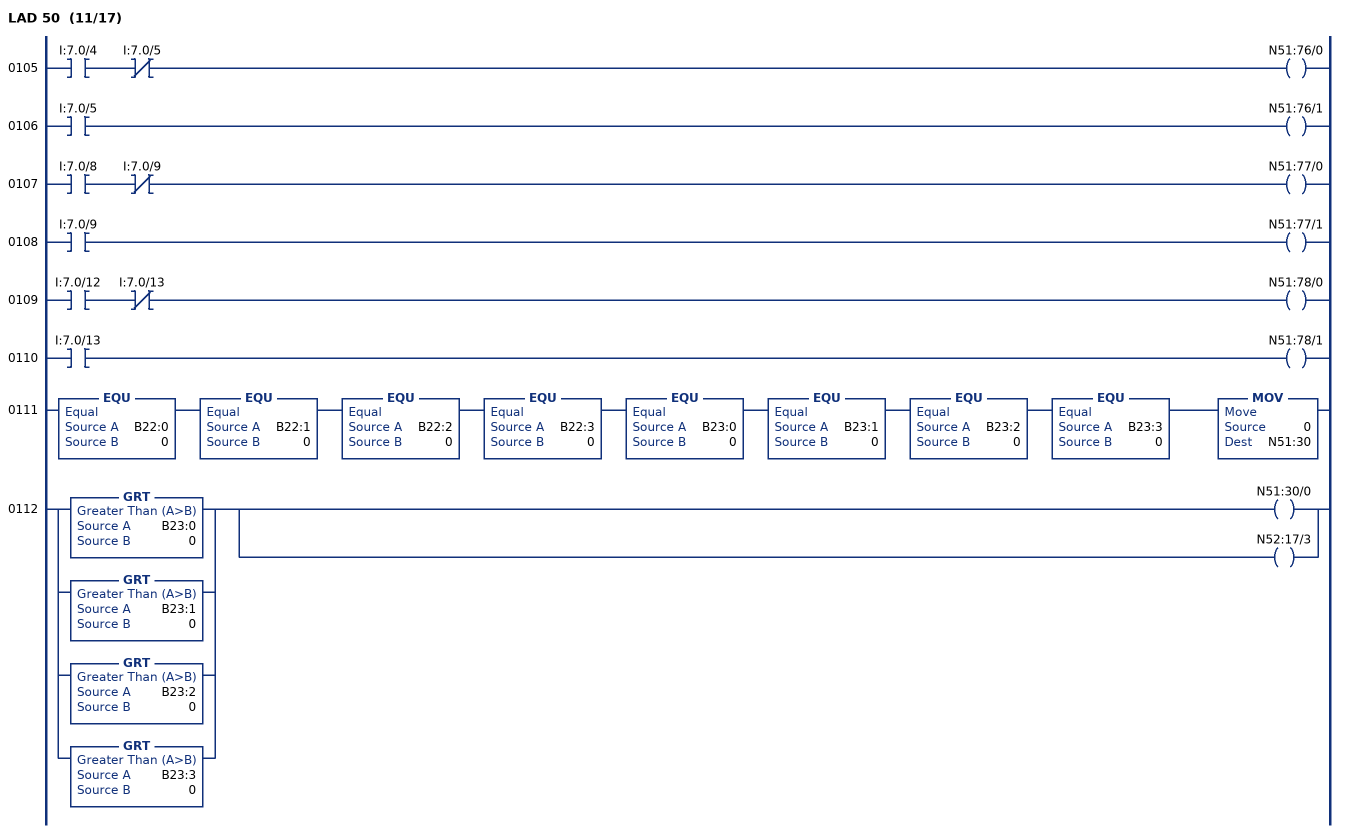
% Rung: 105 %
SOR XIC I:7.0/4 XIO I:7.0/5 OTE N51:76/0 EOR
% Rung: 106 %
SOR XIC I:7.0/5 OTE N51:76/1 EOR
% Rung: 107 %
SOR XIC I:7.0/8 XIO I:7.0/9 OTE N51:77/0 EOR
% Rung: 108 %
SOR XIC I:7.0/9 OTE N51:77/1 EOR
% Rung: 109 %
SOR XIC I:7.0/12 XIO I:7.0/13 OTE N51:78/0 EOR
% Rung: 110 %
SOR XIC I:7.0/13 OTE N51:78/1 EOR
% Rung: 111 %
SOR EQU B22:0 0 EQU B22:1 0 EQU B22:2 0 EQU B22:3 0 EQU B23:0 0 EQU B23:1 0 EQU B23:2 0 EQU B23:3 0 MOV 0 N51:30 EOR
% Rung: 112 %
SOR BST GRT B23:0 0 NXB GRT B23:1 0 NXB GRT B23:2 0 NXB GRT B23:3 0 BND BST OTE N51:30/0 NXB OTE N52:17/3 BND EOR

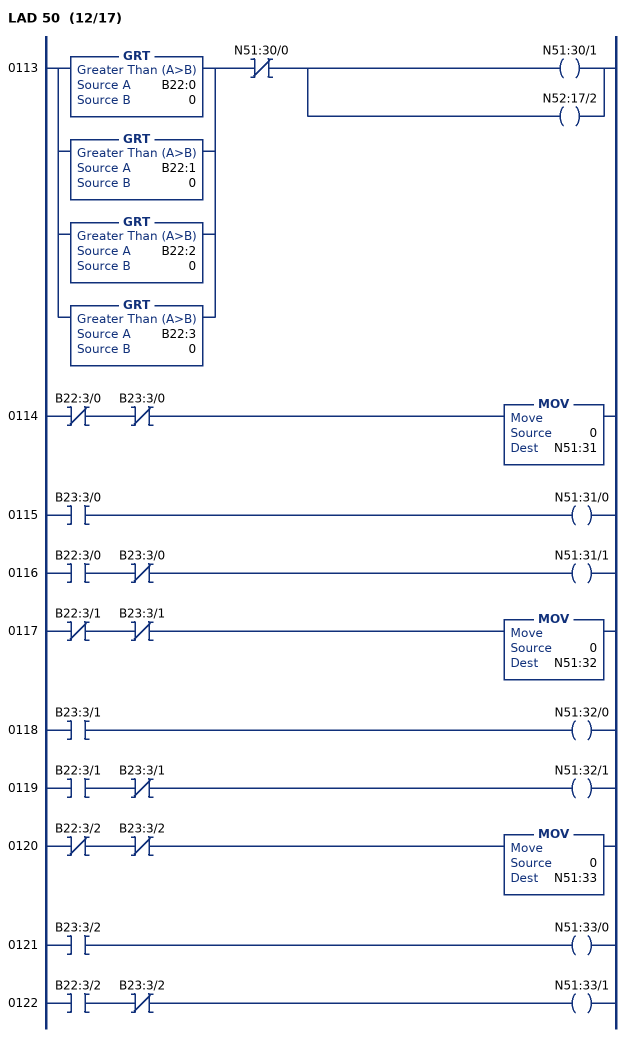
% Rung: 113 %
SOR BST GRT B22:0 0 NXB GRT B22:1 0 NXB GRT B22:2 0 NXB GRT B22:3 0 BND XIO N51:30/0 BST OTE N51:30/1 NXB OTE N52:17/2 BND EOR
% Rung: 114 %
SOR XIO B22:3/0 XIO B23:3/0 MOV 0 N51:31 EOR
% Rung: 115 %
SOR XIC B23:3/0 OTE N51:31/0 EOR
% Rung: 116 %
SOR XIC B22:3/0 XIO B23:3/0 OTE N51:31/1 EOR
% Rung: 117 %
SOR XIO B22:3/1 XIO B23:3/1 MOV 0 N51:32 EOR
% Rung: 118 %
SOR XIC B23:3/1 OTE N51:32/0 EOR
% Rung: 119 %
SOR XIC B22:3/1 XIO B23:3/1 OTE N51:32/1 EOR
% Rung: 120 %
SOR XIO B22:3/2 XIO B23:3/2 MOV 0 N51:33 EOR
% Rung: 121 %
SOR XIC B23:3/2 OTE N51:33/0 EOR
% Rung: 122 %
SOR XIC B22:3/2 XIO B23:3/2 OTE N51:33/1 EOR

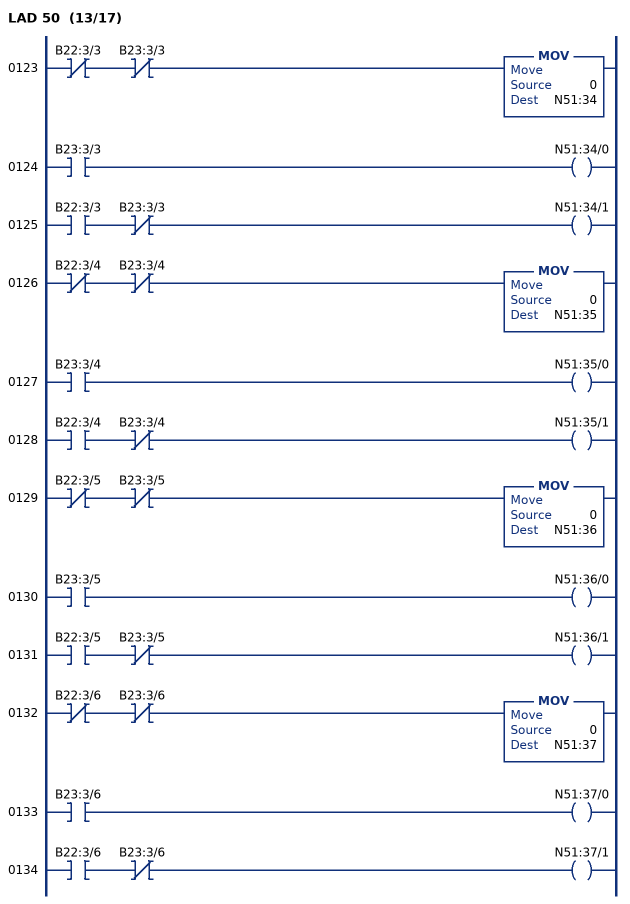
% Rung: 123 %
SOR XIO B22:3/3 XIO B23:3/3 MOV 0 N51:34 EOR
% Rung: 124 %
SOR XIC B23:3/3 OTE N51:34/0 EOR
% Rung: 125 %
SOR XIC B22:3/3 XIO B23:3/3 OTE N51:34/1 EOR
% Rung: 126 %
SOR XIO B22:3/4 XIO B23:3/4 MOV 0 N51:35 EOR
% Rung: 127 %
SOR XIC B23:3/4 OTE N51:35/0 EOR
% Rung: 128 %
SOR XIC B22:3/4 XIO B23:3/4 OTE N51:35/1 EOR
% Rung: 129 %
SOR XIO B22:3/5 XIO B23:3/5 MOV 0 N51:36 EOR
% Rung: 130 %
SOR XIC B23:3/5 OTE N51:36/0 EOR
% Rung: 131 %
SOR XIC B22:3/5 XIO B23:3/5 OTE N51:36/1 EOR
% Rung: 132 %
SOR XIO B22:3/6 XIO B23:3/6 MOV 0 N51:37 EOR
% Rung: 133 %
SOR XIC B23:3/6 OTE N51:37/0 EOR
% Rung: 134 %
SOR XIC B22:3/6 XIO B23:3/6 OTE N51:37/1 EOR

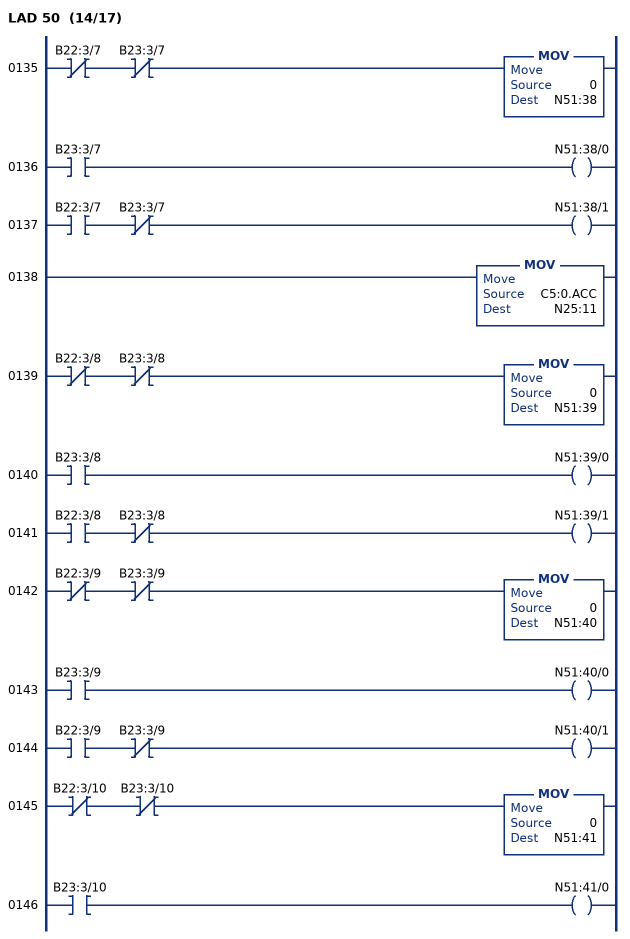
% Rung: 135 %
SOR XIO B22:3/7 XIO B23:3/7 MOV 0 N51:38 EOR
% Rung: 136 %
SOR XIC B23:3/7 OTE N51:38/0 EOR
% Rung: 137 %
SOR XIC B22:3/7 XIO B23:3/7 OTE N51:38/1 EOR
% Rung: 138 %
SOR MOV C5:0.ACC N25:11 EOR
% Rung: 139 %
SOR XIO B22:3/8 XIO B23:3/8 MOV 0 N51:39 EOR
% Rung: 140 %
SOR XIC B23:3/8 OTE N51:39/0 EOR
% Rung: 141 %
SOR XIC B22:3/8 XIO B23:3/8 OTE N51:39/1 EOR
% Rung: 142 %
SOR XIO B22:3/9 XIO B23:3/9 MOV 0 N51:40 EOR
% Rung: 143 %
SOR XIC B23:3/9 OTE N51:40/0 EOR
% Rung: 144 %
SOR XIC B22:3/9 XIO B23:3/9 OTE N51:40/1 EOR
% Rung: 145 %
SOR XIO B22:3/10 XIO B23:3/10 MOV 0 N51:41 EOR
% Rung: 146 %
SOR XIC B23:3/10 OTE N51:41/0 EOR

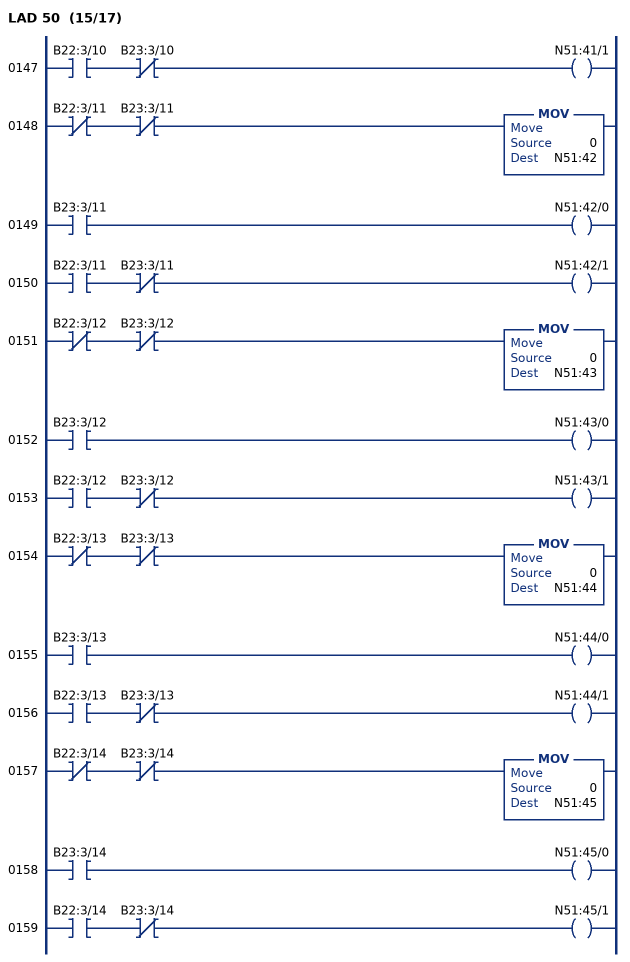
% Rung: 147 %
SOR XIC B22:3/10 XIO B23:3/10 OTE N51:41/1 EOR
% Rung: 148 %
SOR XIO B22:3/11 XIO B23:3/11 MOV 0 N51:42 EOR
% Rung: 149 %
SOR XIC B23:3/11 OTE N51:42/0 EOR
% Rung: 150 %
SOR XIC B22:3/11 XIO B23:3/11 OTE N51:42/1 EOR
% Rung: 151 %
SOR XIO B22:3/12 XIO B23:3/12 MOV 0 N51:43 EOR
% Rung: 152 %
SOR XIC B23:3/12 OTE N51:43/0 EOR
% Rung: 153 %
SOR XIC B22:3/12 XIO B23:3/12 OTE N51:43/1 EOR
% Rung: 154 %
SOR XIO B22:3/13 XIO B23:3/13 MOV 0 N51:44 EOR
% Rung: 155 %
SOR XIC B23:3/13 OTE N51:44/0 EOR
% Rung: 156 %
SOR XIC B22:3/13 XIO B23:3/13 OTE N51:44/1 EOR
% Rung: 157 %
SOR XIO B22:3/14 XIO B23:3/14 MOV 0 N51:45 EOR
% Rung: 158 %
SOR XIC B23:3/14 OTE N51:45/0 EOR
% Rung: 159 %
SOR XIC B22:3/14 XIO B23:3/14 OTE N51:45/1 EOR

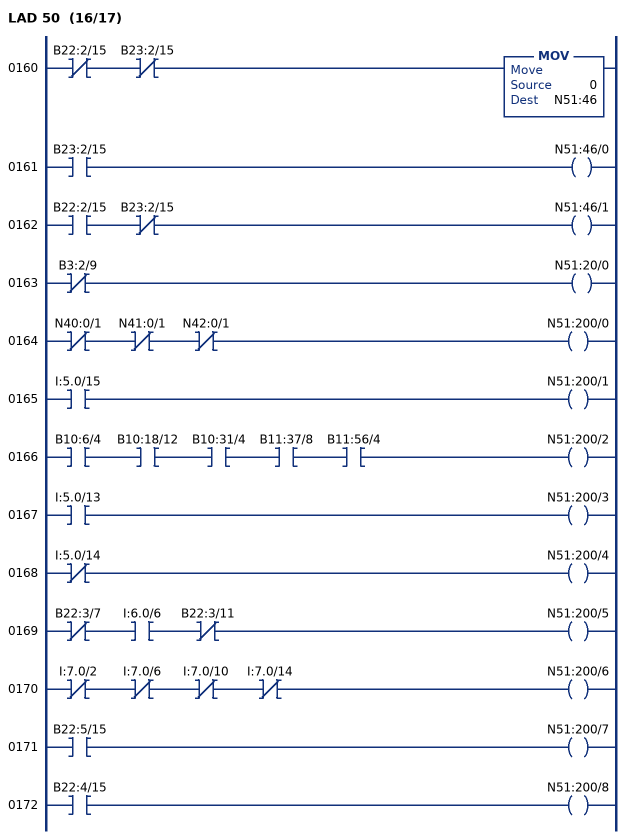
% Rung: 160 %
SOR XIO B22:2/15 XIO B23:2/15 MOV 0 N51:46 EOR
% Rung: 161 %
SOR XIC B23:2/15 OTE N51:46/0 EOR
% Rung: 162 %
SOR XIC B22:2/15 XIO B23:2/15 OTE N51:46/1 EOR
% Rung: 163 %
SOR XIO B3:2/9 OTE N51:20/0 EOR
% Rung: 164 %
SOR XIO N40:0/1 XIO N41:0/1 XIO N42:0/1 OTE N51:200/0 EOR
% Rung: 165 %
SOR XIC I:5.0/15 OTE N51:200/1 EOR
% Rung: 166 %
SOR XIC B10:6/4 XIC B10:18/12 XIC B10:31/4 XIC B11:37/8 XIC B11:56/4 OTE N51:200/2 EOR
% Rung: 167 %
SOR XIC I:5.0/13 OTE N51:200/3 EOR
% Rung: 168 %
SOR XIO I:5.0/14 OTE N51:200/4 EOR
% Rung: 169 %
SOR XIO B22:3/7 XIC I:6.0/6 XIO B22:3/11 OTE N51:200/5 EOR
% Rung: 170 %
SOR XIO I:7.0/2 XIO I:7.0/6 XIO I:7.0/10 XIO I:7.0/14 OTE N51:200/6 EOR
% Rung: 171 %
SOR XIC B22:5/15 OTE N51:200/7 EOR
% Rung: 172 %
SOR XIC B22:4/15 OTE N51:200/8 EOR

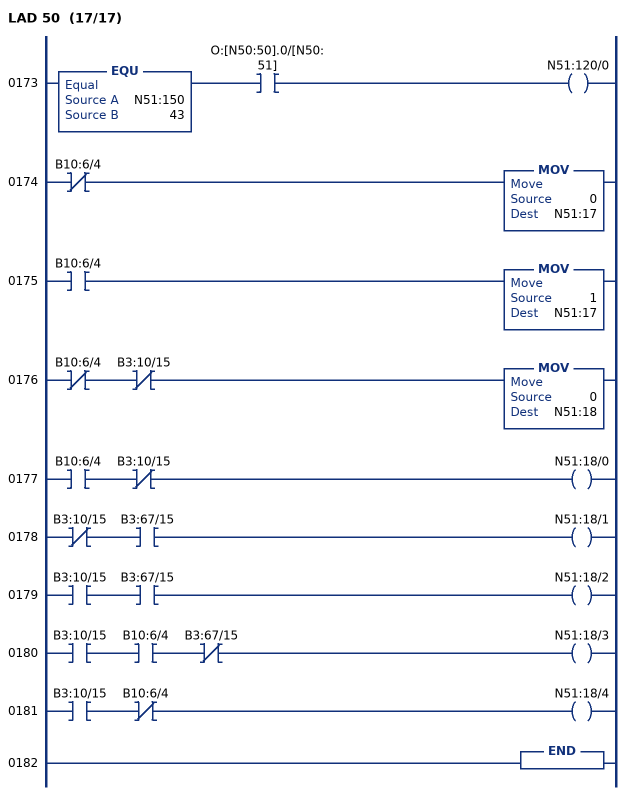
% Rung: 173 %
SOR EQU N51:150 43 XIC O:[N50:50].0/[N50:51] OTE N51:120/0 EOR
% Rung: 174 %
SOR XIO B10:6/4 MOV 0 N51:17 EOR
% Rung: 175 %
SOR XIC B10:6/4 MOV 1 N51:17 EOR
% Rung: 176 %
SOR XIO B10:6/4 XIO B3:10/15 MOV 0 N51:18 EOR
% Rung: 177 %
SOR XIC B10:6/4 XIO B3:10/15 OTE N51:18/0 EOR
% Rung: 178 %
SOR XIO B3:10/15 XIC B3:67/15 OTE N51:18/1 EOR
% Rung: 179 %
SOR XIC B3:10/15 XIC B3:67/15 OTE N51:18/2 EOR
% Rung: 180 %
SOR XIC B3:10/15 XIC B10:6/4 XIO B3:67/15 OTE N51:18/3 EOR
% Rung: 181 %
SOR XIC B3:10/15 XIO B10:6/4 OTE N51:18/4 EOR
% Rung: 182 %
SOR END EOR

LADDER 51
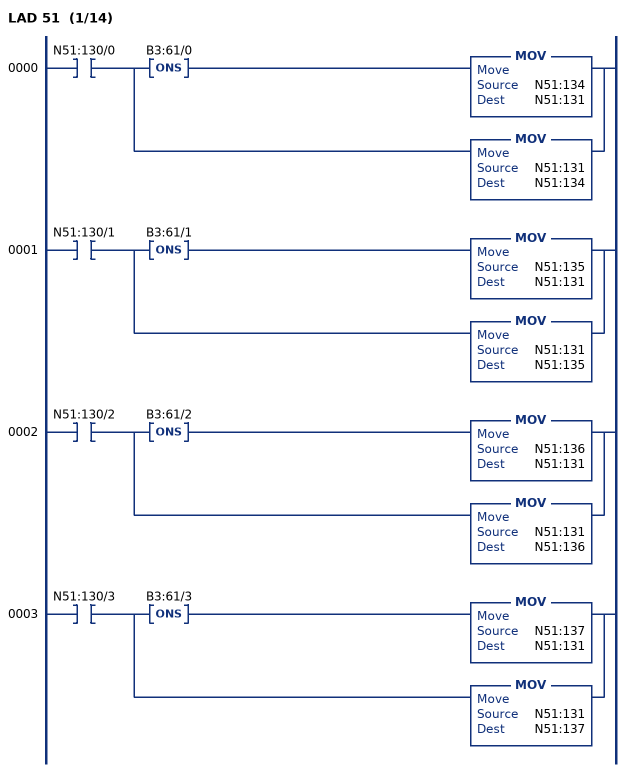
% Rung: 0 %
SOR XIC N51:130/0 BST OSR B3:61/0 MOV N51:134 N51:131 NXB MOV N51:131 N51:134 BND EOR
% Rung: 1 %
SOR XIC N51:130/1 BST OSR B3:61/1 MOV N51:135 N51:131 NXB MOV N51:131 N51:135 BND EOR
% Rung: 2 %
SOR XIC N51:130/2 BST OSR B3:61/2 MOV N51:136 N51:131 NXB MOV N51:131 N51:136 BND EOR
% Rung: 3 %
SOR XIC N51:130/3 BST OSR B3:61/3 MOV N51:137 N51:131 NXB MOV N51:131 N51:137 BND EOR

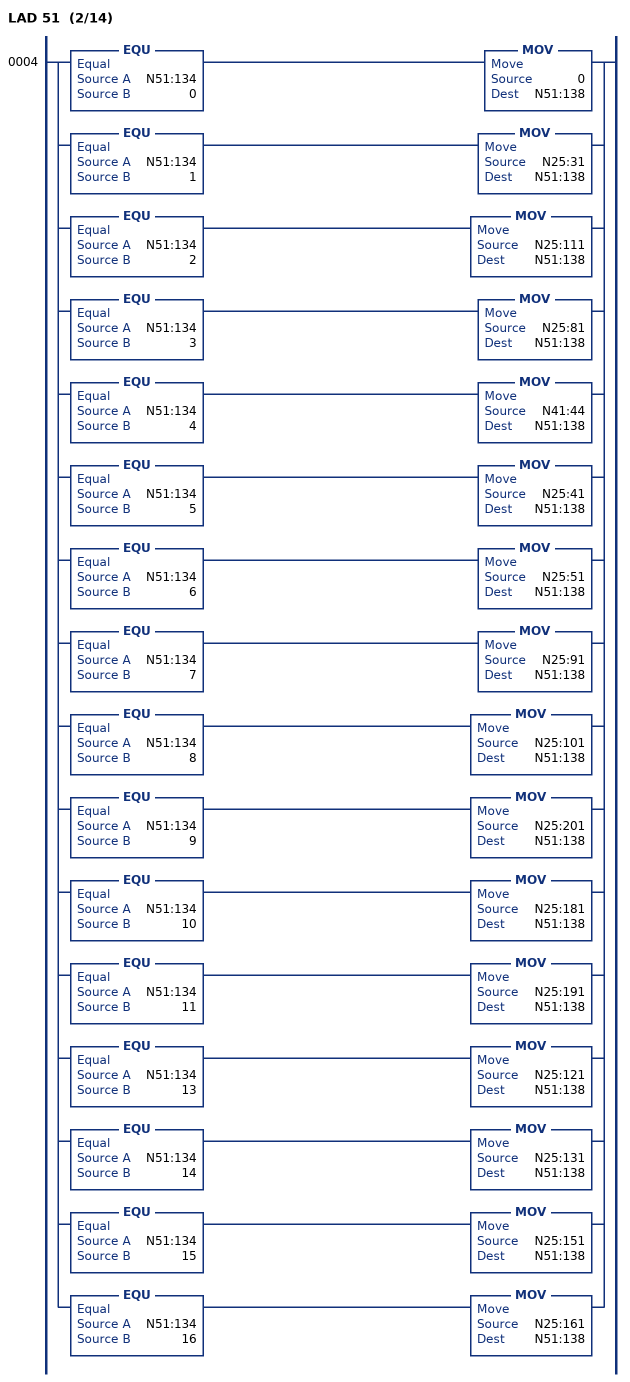
% Rung: 4 %
SOR BST EQU N51:134 0 MOV 0 N51:138 NXB EQU N51:134 1 MOV N25:31 N51:138 NXB EQU N51:134 2 MOV N25:111 N51:138 NXB EQU N51:134 3 MOV N25:81 N51:138 NXB EQU N51:134 4 MOV N41:44 N51:138 NXB EQU N51:134 5 MOV N25:41 N51:138 NXB EQU N51:134 6 MOV N25:51 N51:138 NXB EQU N51:134 7 MOV N25:91 N51:138 NXB EQU N51:134 8 MOV N25:101 N51:138 NXB EQU N51:134 9 MOV N25:201 N51:138 NXB EQU N51:134 10 MOV N25:181 N51:138 NXB EQU N51:134 11 MOV N25:191 N51:138 NXB EQU N51:134 13 MOV N25:121 N51:138 NXB EQU N51:134 14 MOV N25:131 N51:138 NXB EQU N51:134 15 MOV N25:151 N51:138 NXB EQU N51:134 16 MOV N25:161 N51:138 BND EOR

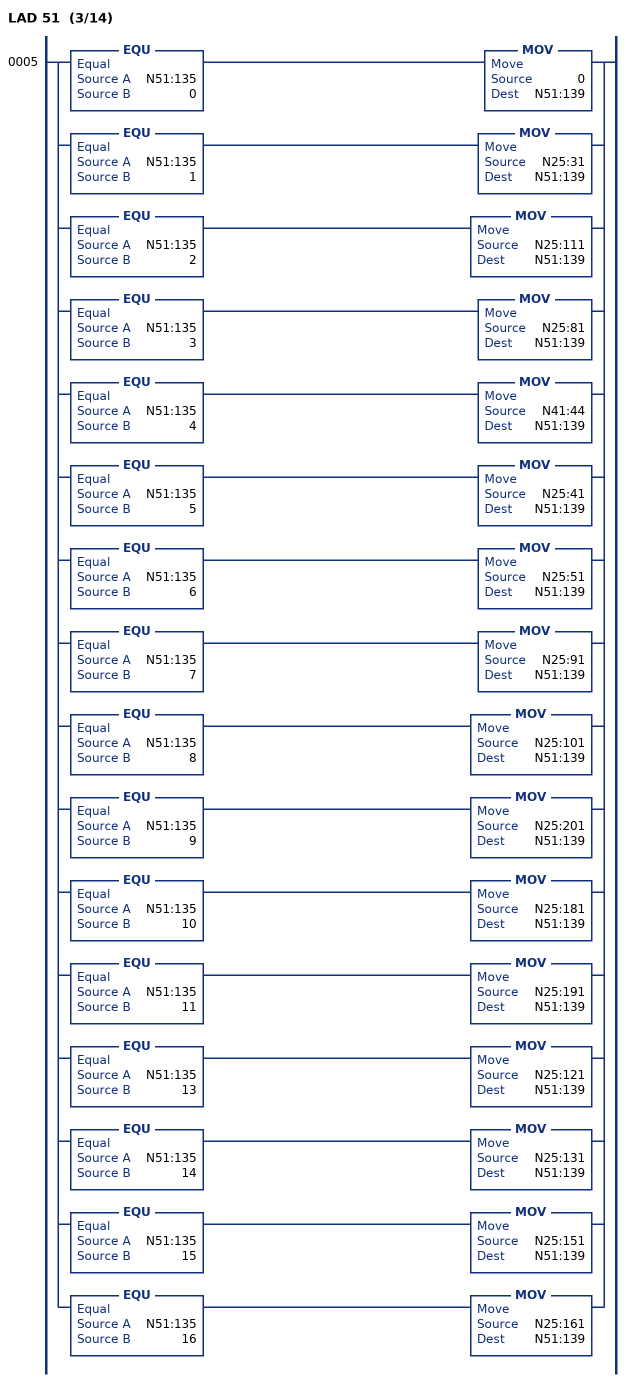
% Rung: 5 %
SOR BST EQU N51:135 0 MOV 0 N51:139 NXB EQU N51:135 1 MOV N25:31 N51:139 NXB EQU N51:135 2 MOV N25:111 N51:139 NXB EQU N51:135 3 MOV N25:81 N51:139 NXB EQU N51:135 4 MOV N41:44 N51:139 NXB EQU N51:135 5 MOV N25:41 N51:139 NXB EQU N51:135 6 MOV N25:51 N51:139 NXB EQU N51:135 7 MOV N25:91 N51:139 NXB EQU N51:135 8 MOV N25:101 N51:139 NXB EQU N51:135 9 MOV N25:201 N51:139 NXB EQU N51:135 10 MOV N25:181 N51:139 NXB EQU N51:135 11 MOV N25:191 N51:139 NXB EQU N51:135 13 MOV N25:121 N51:139 NXB EQU N51:135 14 MOV N25:131 N51:139 NXB EQU N51:135 15 MOV N25:151 N51:139 NXB EQU N51:135 16 MOV N25:161 N51:139 BND EOR

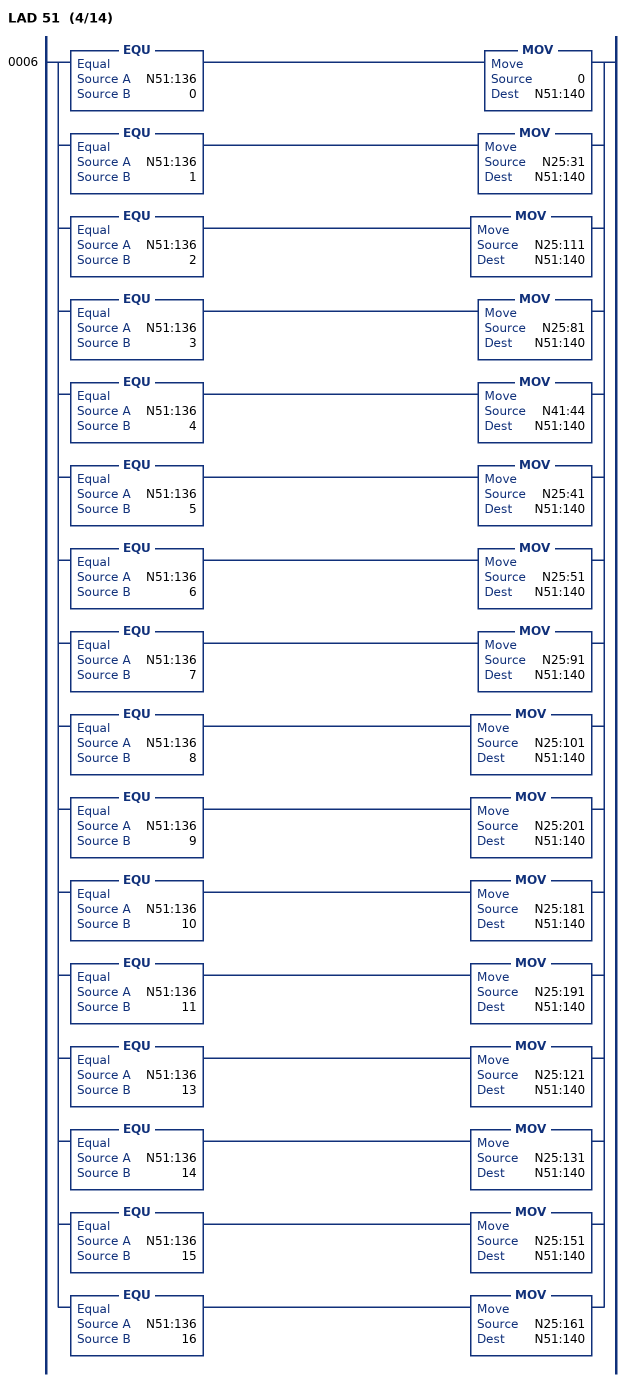
% Rung: 6 %
SOR BST EQU N51:136 0 MOV 0 N51:140 NXB EQU N51:136 1 MOV N25:31 N51:140 NXB EQU N51:136 2 MOV N25:111 N51:140 NXB EQU N51:136 3 MOV N25:81 N51:140 NXB EQU N51:136 4 MOV N41:44 N51:140 NXB EQU N51:136 5 MOV N25:41 N51:140 NXB EQU N51:136 6 MOV N25:51 N51:140 NXB EQU N51:136 7 MOV N25:91 N51:140 NXB EQU N51:136 8 MOV N25:101 N51:140 NXB EQU N51:136 9 MOV N25:201 N51:140 NXB EQU N51:136 10 MOV N25:181 N51:140 NXB EQU N51:136 11 MOV N25:191 N51:140 NXB EQU N51:136 13 MOV N25:121 N51:140 NXB EQU N51:136 14 MOV N25:131 N51:140 NXB EQU N51:136 15 MOV N25:151 N51:140 NXB EQU N51:136 16 MOV N25:161 N51:140 BND EOR

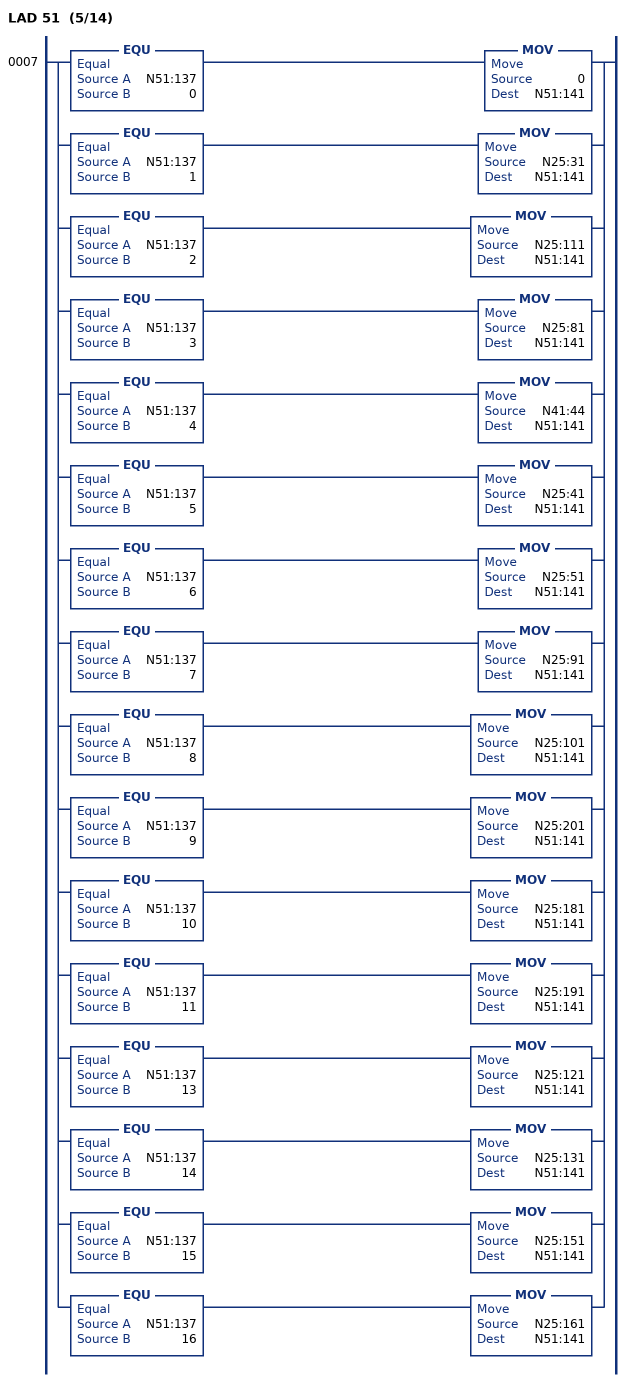
% Rung: 7 %
SOR BST EQU N51:137 0 MOV 0 N51:141 NXB EQU N51:137 1 MOV N25:31 N51:141 NXB EQU N51:137 2 MOV N25:111 N51:141 NXB EQU N51:137 3 MOV N25:81 N51:141 NXB EQU N51:137 4 MOV N41:44 N51:141 NXB EQU N51:137 5 MOV N25:41 N51:141 NXB EQU N51:137 6 MOV N25:51 N51:141 NXB EQU N51:137 7 MOV N25:91 N51:141 NXB EQU N51:137 8 MOV N25:101 N51:141 NXB EQU N51:137 9 MOV N25:201 N51:141 NXB EQU N51:137 10 MOV N25:181 N51:141 NXB EQU N51:137 11 MOV N25:191 N51:141 NXB EQU N51:137 13 MOV N25:121 N51:141 NXB EQU N51:137 14 MOV N25:131 N51:141 NXB EQU N51:137 15 MOV N25:151 N51:141 NXB EQU N51:137 16 MOV N25:161 N51:141 BND EOR

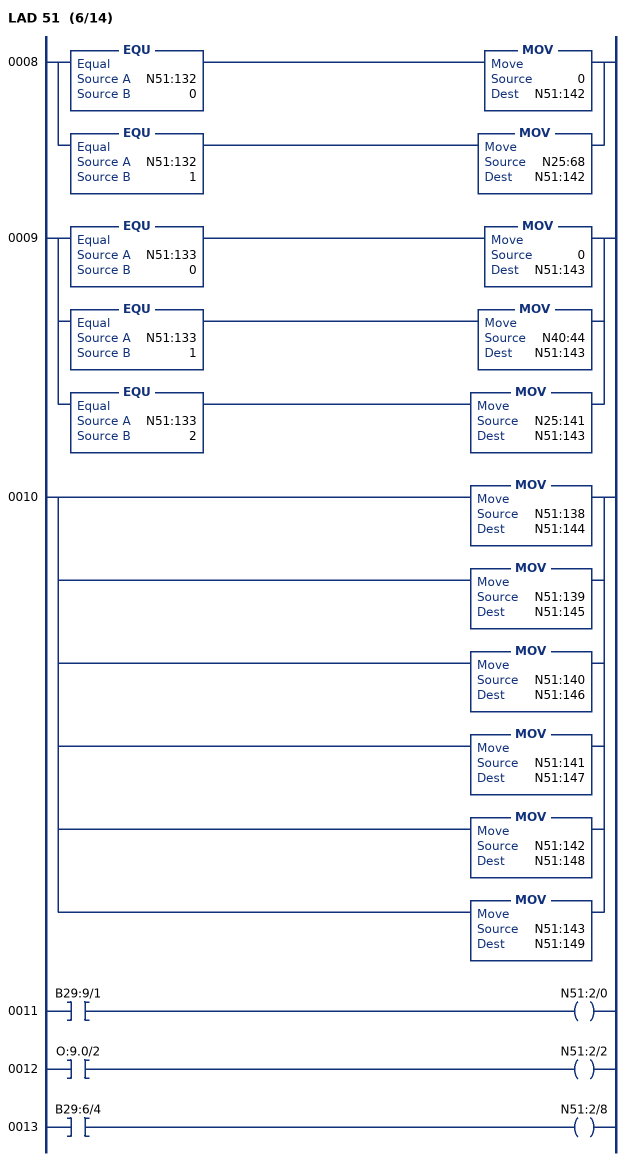
% Rung: 8 %
SOR BST EQU N51:132 0 MOV 0 N51:142 NXB EQU N51:132 1 MOV N25:68 N51:142 BND EOR
% Rung: 9 %
SOR BST EQU N51:133 0 MOV 0 N51:143 NXB EQU N51:133 1 MOV N40:44 N51:143 NXB EQU N51:133 2 MOV N25:141 N51:143 BND EOR
% Rung: 10 %
SOR BST MOV N51:138 N51:144 NXB MOV N51:139 N51:145 NXB MOV N51:140 N51:146 NXB MOV N51:141 N51:147 NXB MOV N51:142 N51:148 NXB MOV N51:143 N51:149 BND EOR
% Rung: 11 %
SOR XIC B29:9/1 OTE N51:2/0 EOR
% Rung: 12 %
SOR XIC O:9.0/2 OTE N51:2/2 EOR
% Rung: 13 %
SOR XIC B29:6/4 OTE N51:2/8 EOR

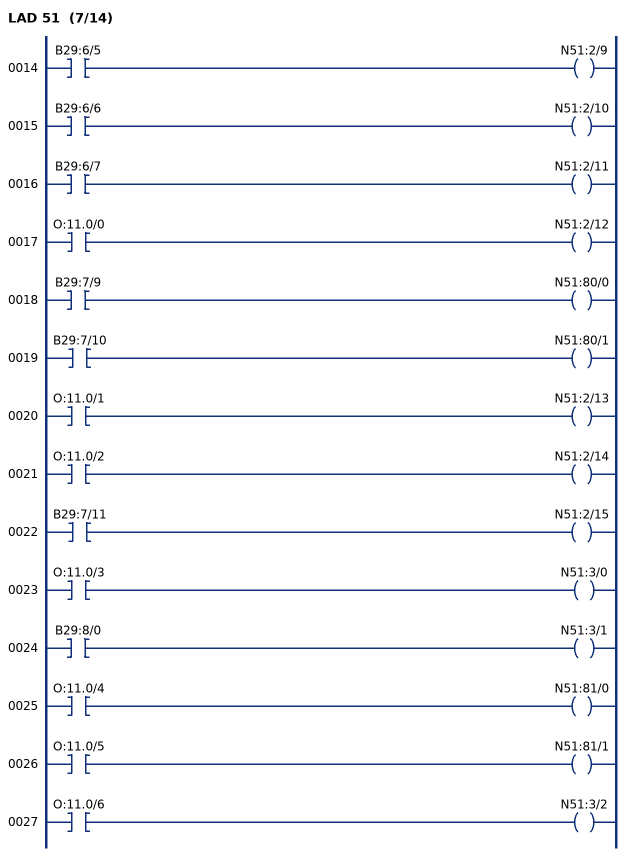
% Rung: 14 %
SOR XIC B29:6/5 OTE N51:2/9 EOR
% Rung: 15 %
SOR XIC B29:6/6 OTE N51:2/10 EOR
% Rung: 16 %
SOR XIC B29:6/7 OTE N51:2/11 EOR
% Rung: 17 %
SOR XIC O:11.0/0 OTE N51:2/12 EOR
% Rung: 18 %
SOR XIC B29:7/9 OTE N51:80/0 EOR
% Rung: 19 %
SOR XIC B29:7/10 OTE N51:80/1 EOR
% Rung: 20 %
SOR XIC O:11.0/1 OTE N51:2/13 EOR
% Rung: 21 %
SOR XIC O:11.0/2 OTE N51:2/14 EOR
% Rung: 22 %
SOR XIC B29:7/11 OTE N51:2/15 EOR
% Rung: 23 %
SOR XIC O:11.0/3 OTE N51:3/0 EOR
% Rung: 24 %
SOR XIC B29:8/0 OTE N51:3/1 EOR
% Rung: 25 %
SOR XIC O:11.0/4 OTE N51:81/0 EOR
% Rung: 26 %
SOR XIC O:11.0/5 OTE N51:81/1 EOR
% Rung: 27 %
SOR XIC O:11.0/6 OTE N51:3/2 EOR

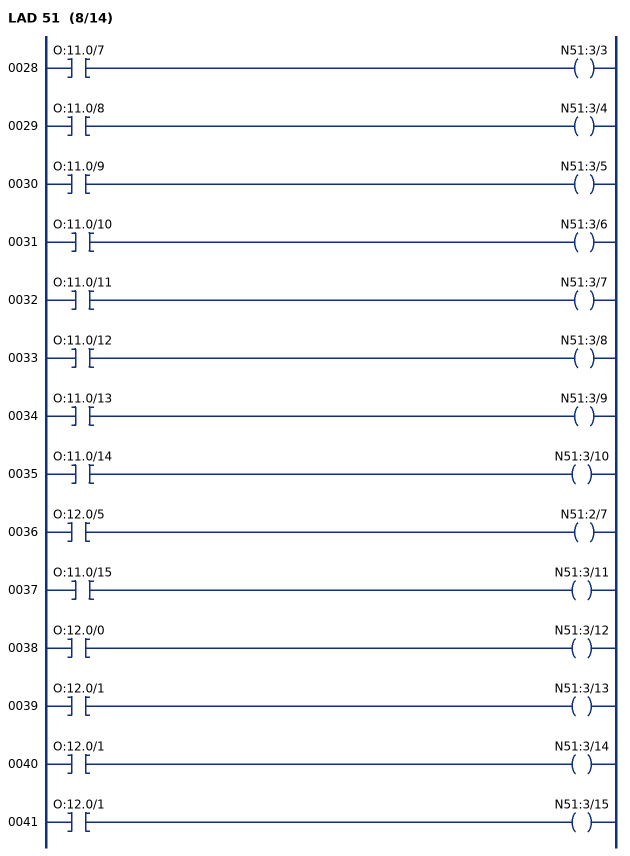
% Rung: 28 %
SOR XIC O:11.0/7 OTE N51:3/3 EOR
% Rung: 29 %
SOR XIC O:11.0/8 OTE N51:3/4 EOR
% Rung: 30 %
SOR XIC O:11.0/9 OTE N51:3/5 EOR
% Rung: 31 %
SOR XIC O:11.0/10 OTE N51:3/6 EOR
% Rung: 32 %
SOR XIC O:11.0/11 OTE N51:3/7 EOR
% Rung: 33 %
SOR XIC O:11.0/12 OTE N51:3/8 EOR
% Rung: 34 %
SOR XIC O:11.0/13 OTE N51:3/9 EOR
% Rung: 35 %
SOR XIC O:11.0/14 OTE N51:3/10 EOR
% Rung: 36 %
SOR XIC O:12.0/5 OTE N51:2/7 EOR
% Rung: 37 %
SOR XIC O:11.0/15 OTE N51:3/11 EOR
% Rung: 38 %
SOR XIC O:12.0/0 OTE N51:3/12 EOR
% Rung: 39 %
SOR XIC O:12.0/1 OTE N51:3/13 EOR
% Rung: 40 %
SOR XIC O:12.0/1 OTE N51:3/14 EOR
% Rung: 41 %
SOR XIC O:12.0/1 OTE N51:3/15 EOR

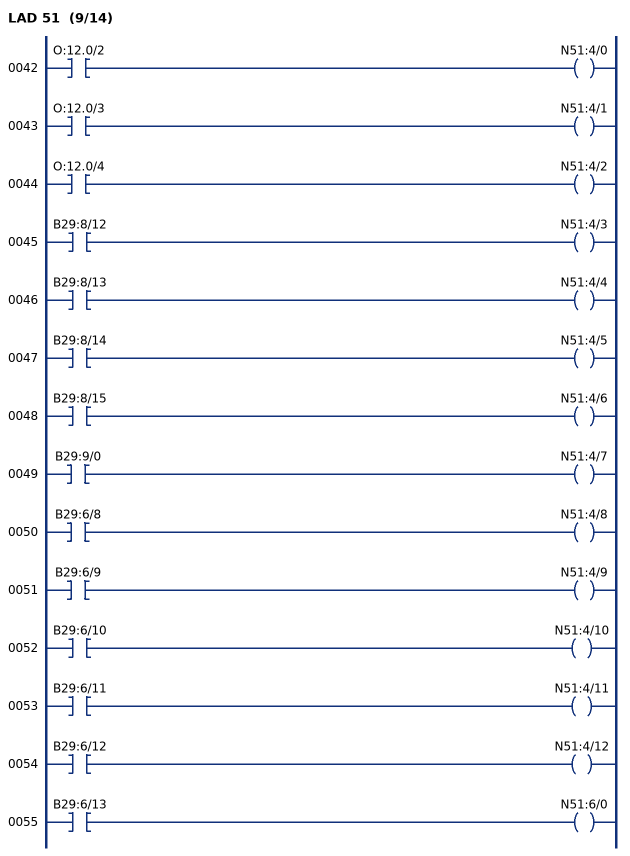
% Rung: 42 %
SOR XIC O:12.0/2 OTE N51:4/0 EOR
% Rung: 43 %
SOR XIC O:12.0/3 OTE N51:4/1 EOR
% Rung: 44 %
SOR XIC O:12.0/4 OTE N51:4/2 EOR
% Rung: 45 %
SOR XIC B29:8/12 OTE N51:4/3 EOR
% Rung: 46 %
SOR XIC B29:8/13 OTE N51:4/4 EOR
% Rung: 47 %
SOR XIC B29:8/14 OTE N51:4/5 EOR
% Rung: 48 %
SOR XIC B29:8/15 OTE N51:4/6 EOR
% Rung: 49 %
SOR XIC B29:9/0 OTE N51:4/7 EOR
% Rung: 50 %
SOR XIC B29:6/8 OTE N51:4/8 EOR
% Rung: 51 %
SOR XIC B29:6/9 OTE N51:4/9 EOR
% Rung: 52 %
SOR XIC B29:6/10 OTE N51:4/10 EOR
% Rung: 53 %
SOR XIC B29:6/11 OTE N51:4/11 EOR
% Rung: 54 %
SOR XIC B29:6/12 OTE N51:4/12 EOR
% Rung: 55 %
SOR XIC B29:6/13 OTE N51:6/0 EOR

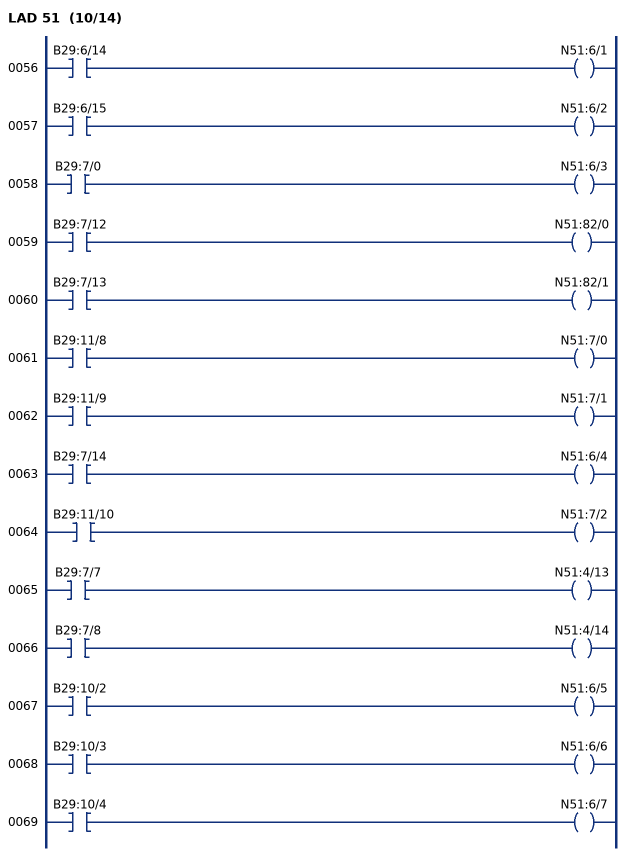
% Rung: 56 %
SOR XIC B29:6/14 OTE N51:6/1 EOR
% Rung: 57 %
SOR XIC B29:6/15 OTE N51:6/2 EOR
% Rung: 58 %
SOR XIC B29:7/0 OTE N51:6/3 EOR
% Rung: 59 %
SOR XIC B29:7/12 OTE N51:82/0 EOR
% Rung: 60 %
SOR XIC B29:7/13 OTE N51:82/1 EOR
% Rung: 61 %
SOR XIC B29:11/8 OTE N51:7/0 EOR
% Rung: 62 %
SOR XIC B29:11/9 OTE N51:7/1 EOR
% Rung: 63 %
SOR XIC B29:7/14 OTE N51:6/4 EOR
% Rung: 64 %
SOR XIC B29:11/10 OTE N51:7/2 EOR
% Rung: 65 %
SOR XIC B29:7/7 OTE N51:4/13 EOR
% Rung: 66 %
SOR XIC B29:7/8 OTE N51:4/14 EOR
% Rung: 67 %
SOR XIC B29:10/2 OTE N51:6/5 EOR
% Rung: 68 %
SOR XIC B29:10/3 OTE N51:6/6 EOR
% Rung: 69 %
SOR XIC B29:10/4 OTE N51:6/7 EOR

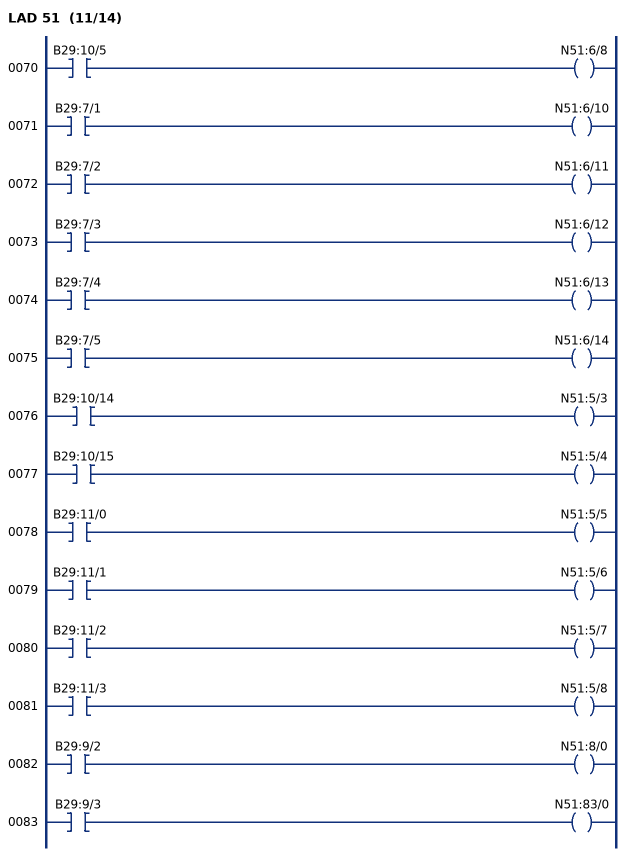
% Rung: 70 %
SOR XIC B29:10/5 OTE N51:6/8 EOR
% Rung: 71 %
SOR XIC B29:7/1 OTE N51:6/10 EOR
% Rung: 72 %
SOR XIC B29:7/2 OTE N51:6/11 EOR
% Rung: 73 %
SOR XIC B29:7/3 OTE N51:6/12 EOR
% Rung: 74 %
SOR XIC B29:7/4 OTE N51:6/13 EOR
% Rung: 75 %
SOR XIC B29:7/5 OTE N51:6/14 EOR
% Rung: 76 %
SOR XIC B29:10/14 OTE N51:5/3 EOR
% Rung: 77 %
SOR XIC B29:10/15 OTE N51:5/4 EOR
% Rung: 78 %
SOR XIC B29:11/0 OTE N51:5/5 EOR
% Rung: 79 %
SOR XIC B29:11/1 OTE N51:5/6 EOR
% Rung: 80 %
SOR XIC B29:11/2 OTE N51:5/7 EOR
% Rung: 81 %
SOR XIC B29:11/3 OTE N51:5/8 EOR
% Rung: 82 %
SOR XIC B29:9/2 OTE N51:8/0 EOR
% Rung: 83 %
SOR XIC B29:9/3 OTE N51:83/0 EOR

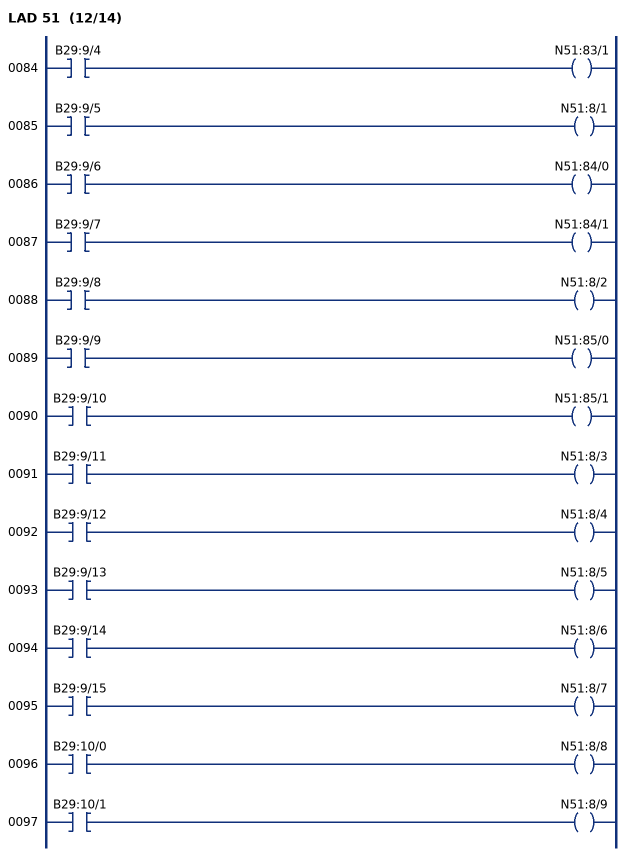
% Rung: 84 %
SOR XIC B29:9/4 OTE N51:83/1 EOR
% Rung: 85 %
SOR XIC B29:9/5 OTE N51:8/1 EOR
% Rung: 86 %
SOR XIC B29:9/6 OTE N51:84/0 EOR
% Rung: 87 %
SOR XIC B29:9/7 OTE N51:84/1 EOR
% Rung: 88 %
SOR XIC B29:9/8 OTE N51:8/2 EOR
% Rung: 89 %
SOR XIC B29:9/9 OTE N51:85/0 EOR
% Rung: 90 %
SOR XIC B29:9/10 OTE N51:85/1 EOR
% Rung: 91 %
SOR XIC B29:9/11 OTE N51:8/3 EOR
% Rung: 92 %
SOR XIC B29:9/12 OTE N51:8/4 EOR
% Rung: 93 %
SOR XIC B29:9/13 OTE N51:8/5 EOR
% Rung: 94 %
SOR XIC B29:9/14 OTE N51:8/6 EOR
% Rung: 95 %
SOR XIC B29:9/15 OTE N51:8/7 EOR
% Rung: 96 %
SOR XIC B29:10/0 OTE N51:8/8 EOR
% Rung: 97 %
SOR XIC B29:10/1 OTE N51:8/9 EOR

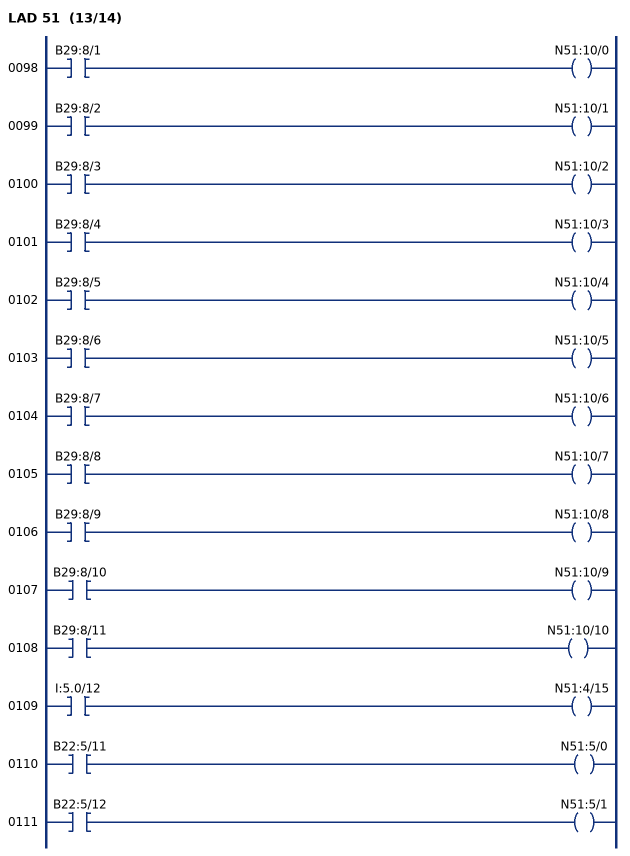
% Rung: 98 %
SOR XIC B29:8/1 OTE N51:10/0 EOR
% Rung: 99 %
SOR XIC B29:8/2 OTE N51:10/1 EOR
% Rung: 100 %
SOR XIC B29:8/3 OTE N51:10/2 EOR
% Rung: 101 %
SOR XIC B29:8/4 OTE N51:10/3 EOR
% Rung: 102 %
SOR XIC B29:8/5 OTE N51:10/4 EOR
% Rung: 103 %
SOR XIC B29:8/6 OTE N51:10/5 EOR
% Rung: 104 %
SOR XIC B29:8/7 OTE N51:10/6 EOR
% Rung: 105 %
SOR XIC B29:8/8 OTE N51:10/7 EOR
% Rung: 106 %
SOR XIC B29:8/9 OTE N51:10/8 EOR
% Rung: 107 %
SOR XIC B29:8/10 OTE N51:10/9 EOR
% Rung: 108 %
SOR XIC B29:8/11 OTE N51:10/10 EOR
% Rung: 109 %
SOR XIC I:5.0/12 OTE N51:4/15 EOR
% Rung: 110 %
SOR XIC B22:5/11 OTE N51:5/0 EOR
% Rung: 111 %
SOR XIC B22:5/12 OTE N51:5/1 EOR

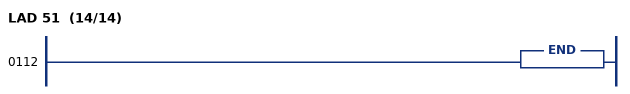
% Rung: 112 %
SOR END EOR

LADDER 52
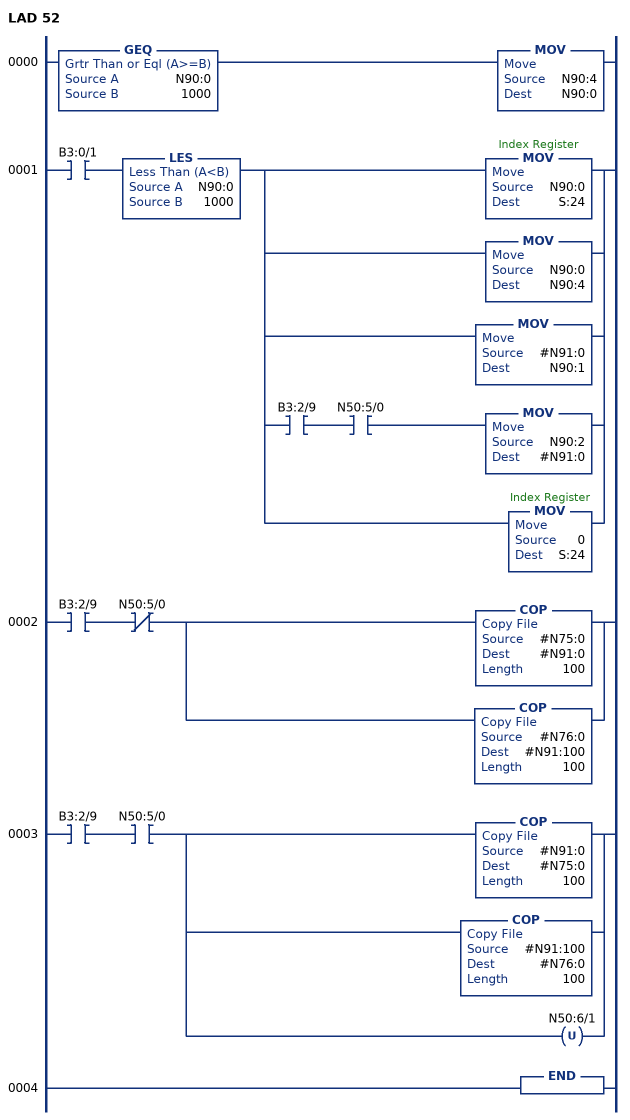
% Rung: 0 %
SOR GEQ N90:0 1000 MOV N90:4 N90:0 EOR
% Rung: 1 %
SOR XIC B3:0/1 LES N90:0 1000 BST MOV N90:0 S:24 NXB MOV N90:0 N90:4 NXB MOV #N91:0 N90:1 NXB XIC B3:2/9 XIC N50:5/0 MOV N90:2 #N91:0 NXB MOV 0 S:24 BND EOR
%   S:24  "Index Register" %
% Rung: 2 %
SOR XIC B3:2/9 XIO N50:5/0 BST COP #N75:0 #N91:0 100 NXB COP #N76:0 #N91:100 100 BND EOR
% Rung: 3 %
SOR XIC B3:2/9 XIC N50:5/0 BST COP #N91:0 #N75:0 100 NXB COP #N91:100 #N76:0 100 NXB OTU N50:6/1 BND EOR
% Rung: 4 %
SOR END EOR

LADDER 53
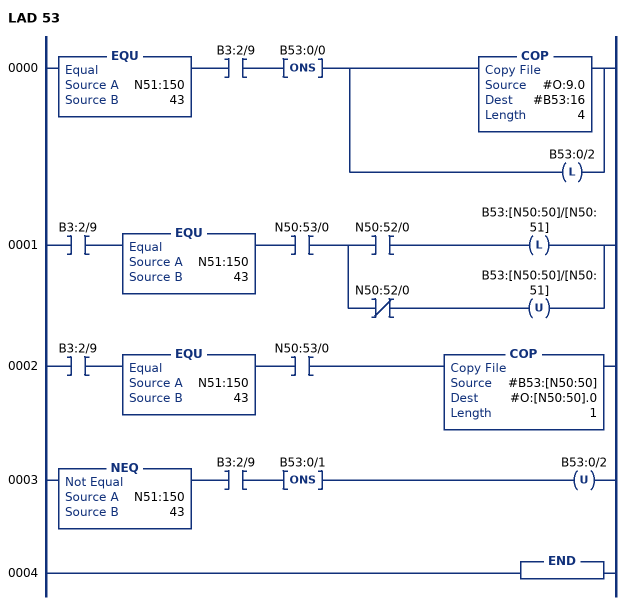
% Rung: 0 %
SOR EQU N51:150 43 XIC B3:2/9 OSR B53:0/0 BST COP #O:9.0 #B53:16 4 NXB OTL B53:0/2 BND EOR
% Rung: 1 %
SOR XIC B3:2/9 EQU N51:150 43 XIC N50:53/0 BST XIC N50:52/0 OTL B53:[N50:50]/[N50:51] NXB XIO N50:52/0 OTU B53:[N50:50]/[N50:51] BND EOR
% Rung: 2 %
SOR XIC B3:2/9 EQU N51:150 43 XIC N50:53/0 COP #B53:[N50:50] #O:[N50:50].0 1 EOR
% Rung: 3 %
SOR NEQ N51:150 43 XIC B3:2/9 OSR B53:0/1 OTU B53:0/2 EOR
% Rung: 4 %
SOR END EOR

LADDER 71
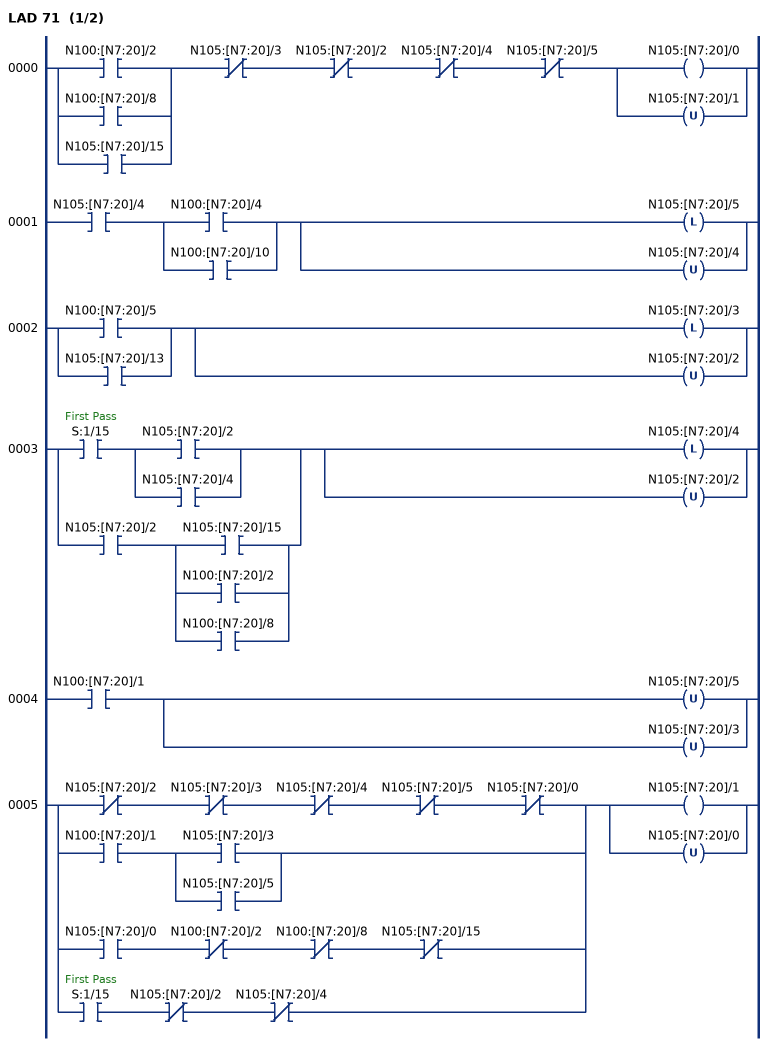
% Rung: 0 %
SOR BST XIC N100:[N7:20]/2 NXB XIC N100:[N7:20]/8 NXB XIC N105:[N7:20]/15 BND XIO N105:[N7:20]/3 XIO N105:[N7:20]/2 XIO N105:[N7:20]/4 XIO N105:[N7:20]/5 BST OTE N105:[N7:20]/0 NXB OTU N105:[N7:20]/1 BND EOR
% Rung: 1 %
SOR XIC N105:[N7:20]/4 BST XIC N100:[N7:20]/4 NXB XIC N100:[N7:20]/10 BND BST OTL N105:[N7:20]/5 NXB OTU N105:[N7:20]/4 BND EOR
% Rung: 2 %
SOR BST XIC N100:[N7:20]/5 NXB XIC N105:[N7:20]/13 BND BST OTL N105:[N7:20]/3 NXB OTU N105:[N7:20]/2 BND EOR
% Rung: 3 %
SOR BST XIC S:1/15 BST XIC N105:[N7:20]/2 NXB XIC N105:[N7:20]/4 BND NXB XIC N105:[N7:20]/2 BST XIC N105:[N7:20]/15 NXB XIC N100:[N7:20]/2 NXB XIC N100:[N7:20]/8 BND BND BST OTL N105:[N7:20]/4 NXB OTU N105:[N7:20]/2 BND EOR
%   S:1/15  "First Pass" %
% Rung: 4 %
SOR XIC N100:[N7:20]/1 BST OTU N105:[N7:20]/5 NXB OTU N105:[N7:20]/3 BND EOR
% Rung: 5 %
SOR BST XIO N105:[N7:20]/2 XIO N105:[N7:20]/3 XIO N105:[N7:20]/4 XIO N105:[N7:20]/5 XIO N105:[N7:20]/0 NXB XIC N100:[N7:20]/1 BST XIC N105:[N7:20]/3 NXB XIC N105:[N7:20]/5 BND NXB XIC N105:[N7:20]/0 XIO N100:[N7:20]/2 XIO N100:[N7:20]/8 XIO N105:[N7:20]/15 NXB XIC S:1/15 XIO N105:[N7:20]/2 XIO N105:[N7:20]/4 BND BST OTE N105:[N7:20]/1 NXB OTU N105:[N7:20]/0 BND EOR
%   S:1/15  "First Pass" %

